// TIA Portal V21 export
DATA_BLOCK "Gestione_010102"   // DB12
{ S7_Optimized_Access := 'TRUE' }
// stored: MemoryReserve 100
   VAR RETAIN
      ComandoRecupero_MemoPulsante : Bool := FALSE;
      ComandoRecupero_Stato : Bool := TRUE;
      RichiestaProdotto_Mostra : Bool := TRUE;
      RichiestaProdotto_ConfermataHmi : Bool := TRUE;
      RichiestaProdotto_Out : Bool := TRUE;
      AbilitazioneProduzione : Bool := TRUE;
      TerminaProduzione : Bool := FALSE;
      TerminaProduzione_Mostra : Bool := TRUE;
      MetricubiTubazioneRiempimento : Real := 1.0;
      MetricubiTubazioneSvuotamento : Real := 0.9;
   END_VAR
   VAR
      AperturaContropressioneFiltri : Real := 100.0;
   END_VAR
BEGIN
END_DATA_BLOCK
